FUNCTION_BLOCK fb_discrete_pi

VAR_INPUT
	// signal inputs
	set_point: REAL := 0.0;
	xmeas_in: REAL := 0.0;
	
	// parameters
	kc: REAL;
	ti: REAL;
	ts: REAL;
	hi: REAL := 100;
	lo: REAL;
	x0: REAL;
		
END_VAR

VAR_OUTPUT
	yout: REAL; // needs to be initialized by caller
END_VAR

VAR
	vel_pi: fb_vel_pi := (kc:=kc, ti:=ti, ts:=ts);
	dpi_unit_delay: fb_unitdelay_real := (xlast:=x0);
END_VAR

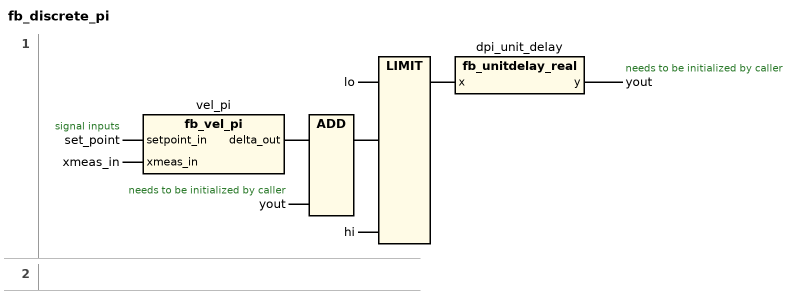
// NETWORK 1
//   set_point: signal inputs
//   yout: needs to be initialized by caller
vel_pi(setpoint_in := set_point, xmeas_in := xmeas_in); // fb_vel_pi
dpi_unit_delay(x := LIMIT(lo, vel_pi.delta_out + yout, hi)); // fb_unitdelay_real
yout := dpi_unit_delay.y;

// NETWORK 2

END_FUNCTION_BLOCK

(* stored: Version 1.1.0.1, ProductVersion 3.1.0.26
   POU fb_discrete_pi: Id {bb2380db-fdca-47e9-9e4d-57d047ddd25f} *)
